Staubli VAL3: getPtPara.pgx

program getPtPara(string x_sPtPara, string& x_sOutPtpara[])
  local num l_nRes
  local num l_ni
begin
  //对参数x_sPtPara进行解析，得到相应信息
  //x_sPtPara结构：p1/p2/IO1/IO2/0.1
  //若没有，使用-1代替
  call PublicProg:SplitChar(l_nRes,x_sPtPara,"/",x_sOutPtpara)

end
